{attribute 'qualified_only'}
VAR_GLOBAL
	//input
	PB1: BOOL;
	PB2: BOOL;
	PBE: BOOL;
	PS1: BOOL;
	PS2: BOOL;
	PS3: BOOL;
	PS4: BOOL;
	PS5: BOOL;
	CS_BIANCO: BOOL;
	CS_NERO: BOOL;
	
	//output
	L1: BOOL;
	L2: BOOL;
	L3: BOOL;
	L4: BOOL;
	L5: BOOL;
	M1 : BOOL;
	M2 : BOOL;
	M3 : BOOL;
	M4 : BOOL;
	M5 : BOOL;
	P1 : BOOL;
	P2 : BOOL;
	P3 : BOOL;
	P4 : BOOL;
END_VAR

(* stored: Version 1.1.0.1, ProductVersion 3.1.4024.12
   GVL GVL: Id {a6c4ee90-e200-4b0b-bf67-f648e428f6e8} *)
